Universal Robots PolyScope program: adaptiveGripper.urp

Program adaptiveGripper (installation=20240827 directory=/programs/show createdIn=5.15.1 lastSavedIn=5.15.1 robotSerialNumber=20245500285)
Calibrated DH parameters: a=[0.000097, -0.210459, -0.026602, 0.000137, 0.000078, 0]; d=[0.162601, 254.180657, -54.076236, -199.970743, 0.099615, 0.099684]; alpha=[1.569796, -0.001455, 0.001957, 1.570525, -1.571561, 0]; deltaTheta=[0, -1.053331, 8.839472, -1.50296, 0.000002, 0]
InitVariablesNode
Robot Program (runOnlyOnce=false)
  MoveL speed 250 mm/s, acceleration 1200 mm/s^2 (useActiveTCP=true) feature=Base
    SuppressedNode
      Waypoint 路点_3: TCP in base x=369.973 y=-402.554 z=99.436 mm, rx=0.2839 ry=2.472 rz=-0.0522 rad; joints [98.977, -86.49, 132.031, -149.747, -54.987, 26.732] deg; TCP offset x=-0.17 y=0 z=192.95 mm, rx=0 ry=0 rz=0 rad
    Waypoint 路点_5: TCP in base x=342.172 y=-354.718 z=152.149 mm, rx=-0.1974 ry=2.8241 rz=-0.0445 rad; joints [107.568, -95.738, 120.747, -121.185, -73.204, 10.644] deg
    SuppressedNode
      Waypoint 路点_6: TCP in base x=599.294 y=-316.459 z=207.229 mm, rx=-0.1973 ry=2.8241 rz=-0.0445 rad; joints [135.376, -75.011, 91.412, -119.77, -78.011, 38.977] deg
  If False
    MoveL speed 250 mm/s, acceleration 1200 mm/s^2 (useActiveTCP=true) feature=Base
      Waypoint 路点_4: TCP in base x=299.736 y=-241.589 z=43.037 mm, rx=-0.0909 ry=3.1401 rz=-0.0002 rad; joints [120.706, -95.486, 135.151, -129.72, -90.042, 27.529] deg
  x := 0.04
  y := 0.03
  yy := 0.06
  z := 0.01
  zegg := -0.025
  h := 0.05
  base := pose_add(路点_4, p[0,0,0.01,0,0,0])
  'egg left'
  var_1 := base
  Script: var_1[0]=var_1[0]-0.04
  Script: var_1[1]=var_1[1]-0.06
  'egg right'
  var_2 := base
  Script: var_2[0]=var_2[0]-0.04
  Script: var_2[1]=var_2[1]+0.06
  'egg'
  var_3 := base
  Script: var_3[0]=var_3[0]-0.04
  Script: var_3[2]=var_3[2]-0.035
  'left'
  var_4 := base
  Script: var_4[0]=var_4[0]+0.04
  Script: var_4[1]=var_4[1]-0.05
  Script: var_4[2]=var_4[2]-0.01
  'right 1'
  var_5 := base
  Script: var_5[0]=var_5[0]+0.04
  Script: var_5[1]=var_5[1]+0.02
  Script: var_5[2]=var_5[2]-0.01
  'right 2'
  var_6 := base
  Script: var_6[0]=var_6[0]+0.02
  Script: var_6[1]=var_6[1]+0.06
  obj := [var_1,var_2,var_3,var_4,var_6,var_5]
  n := 0
  Script: usb = rpc_factory("xmlrpc","http://192.168.1.7:9120/RPC2")
  Script: usb.open()
  Loop Forever
    Popup Message (haltProgram=false message=12 inputType=Text)
    Script: usb.adaptiveClose()
    Wait Sleep waitTime=0.3
    If n≟5
      Popup Message (haltProgram=false message=12 inputType=Text)
      Script: usb.open()
      Popup Message (haltProgram=false message=12 inputType=Text)
      Script: usb.adaptiveClose()
    target := obj[n]
    If n≟2
      before_target := pose_add(target, p[0,0,0.02,0,0,0])
      MoveJ speed 180 deg/s, acceleration 1000 deg/s^2 (useActiveTCP=true) feature=Base
        Waypoint Variable (Variable): variable(name=before_target)
    MoveJ speed 180 deg/s, acceleration 1000 deg/s^2 (useActiveTCP=true) feature=Base
      Waypoint Variable (Variable): variable(name=target)
    Wait Sleep waitTime=0.1
    Script: usb.open()
    If n≟2
      before_target := pose_add(target, p[0,0,0.04,0,0,0])
      MoveJ speed 180 deg/s, acceleration 1000 deg/s^2 (useActiveTCP=true) feature=Base
        Waypoint Variable (Variable): variable=before_target
      SuppressedNode
        Popup Message (haltProgram=false message=xc inputType=Text)
    MoveJ speed 180 deg/s, acceleration 1000 deg/s^2 (useActiveTCP=true) feature=Base
      SuppressedNode
        Waypoint 路点_3: TCP in base x=369.973 y=-402.554 z=99.436 mm, rx=0.2839 ry=2.472 rz=-0.0522 rad; joints [98.977, -86.49, 132.031, -149.747, -54.987, 26.732] deg
      Waypoint 路点_5: TCP in base x=342.172 y=-354.718 z=152.149 mm, rx=-0.1974 ry=2.8241 rz=-0.0445 rad; joints [107.568, -95.738, 120.747, -121.185, -73.204, 10.644] deg
      SuppressedNode
        Waypoint 路点_6: TCP in base x=599.294 y=-316.459 z=207.229 mm, rx=-0.1973 ry=2.8241 rz=-0.0445 rad; joints [135.376, -75.011, 91.412, -119.77, -78.011, 38.977] deg
    Script: n=n+1
    If n≥6
      n := 0
  Halt
  MoveJ speed 60 deg/s, acceleration 80 deg/s^2 (useActiveTCP=true) feature=Base
    SuppressedNode
      Waypoint home: TCP in base x=299.73 y=-241.579 z=97.861 mm, rx=-0.091 ry=3.1401 rz=-0.0002 rad; joints [120.708, -101.14, 130.022, -118.935, -90.022, 27.531] deg
    Waypoint 路点_4 referenceName=路点_4: TCP in base x=299.736 y=-241.589 z=43.037 mm, rx=-0.0909 ry=3.1401 rz=-0.0002 rad; joints [120.706, -95.486, 135.151, -129.72, -90.042, 27.529] deg
    tcpxy := pose_add(路点_4, p[x,y,z,0,0,0])
    tcpxyzzz := pose_add(tcpxy, p[0,0,h,0,0,0])
    varx_y := pose_add(路点_4, p[x,-y,z,0,0,0])
    var_x_y := pose_add(路点_4, p[-x,-yy,z,0,0,0])
    tcp_xy := pose_add(路点_4, p[-x,yy,z,0,0,0])
    tcpegg := pose_add(路点_4, p[-x,0,zegg,0,0,0])
    Waypoint Variable (Variable): variable(name=tcpxyzzz)
    Waypoint Variable (Variable): variable(name=tcpxy)
    Waypoint Variable (Variable): variable(name=varx_y)
    Waypoint Variable (Variable): variable(name=var_x_y)
    Waypoint Variable (Variable): variable(name=tcp_xy)
    Waypoint Variable (Variable): variable(name=tcpegg)
    Popup Message (haltProgram=false message=00 inputType=Text)
  MoveL speed 250 mm/s, acceleration 1200 mm/s^2 (useActiveTCP=true) feature=Base
    x := 0.03
    zegg := -0.025
    tcpegg := pose_add(路点_4, p[-x,0,zegg,0,0,0])
    Waypoint Variable (Variable): variable=tcpegg
  Loop Forever
    Script: usb.open()
    SuppressedNode
      Wait Sleep waitTime=0.5
    Popup Message (haltProgram=false message=12 inputType=Text)
    SuppressedNode
      MoveJ speed 60 deg/s, acceleration 80 deg/s^2 (useActiveTCP=true) feature=Base
        SuppressedNode
          Waypoint 路点_1: TCP in base x=191.611 y=-565.461 z=6.817 mm, rx=-2.2765 ry=-2.1528 rz=-0.0082 rad; joints [95.723, -64.864, 103.956, -128.576, -90.128, 99.099] deg
    Script: usb.adaptiveClose()
    SuppressedNode
      Wait Sleep waitTime=0.5
    SuppressedNode
      MoveL speed 250 mm/s, acceleration 1200 mm/s^2 (useActiveTCP=true) feature=Base
        Waypoint 路点_2: TCP in base x=191.566 y=-565.44 z=47.246 mm, rx=-2.2766 ry=-2.1527 rz=-0.0083 rad; joints [95.72, -68.174, 101.706, -123.011, -90.114, 99.104] deg
    SuppressedNode
      MoveJ speed 60 deg/s, acceleration 80 deg/s^2 (useActiveTCP=true) feature=Base
        Waypoint 路点_1: TCP in base x=191.611 y=-565.461 z=6.817 mm, rx=-2.2765 ry=-2.1528 rz=-0.0082 rad; joints [95.723, -64.864, 103.956, -128.576, -90.128, 99.099] deg
    Popup Message (haltProgram=false message=12 inputType=Text)
    Script: counter=counter+1
